PROGRAM POUNCPowerOn
VAR
	fbXAxisPowerOn : MC_Power;
	fbXAxisDrive : MC_MoveRelative;
	DegreesToRelativeMovment_0: DegreesToRelativeMovment;
	movementBuffer : MC_BufferMode; 
	SetMaxRelativePoint : LREAL;
	SetMaxSteeringAngle : INT;
	inputAngle : INT;
	ExecuteMovement : BOOL;
	ExecuteMovement1 : BOOL;
	MC_MoveAbsolute_0: MC_MoveAbsolute;
	MC_Home_0: MC_Home;
	StartHoming: BOOL;
	endSW AT %I*: BOOL;
	HomingActive: BOOL;
	MC_Reset_0: MC_Reset;
	reset: BOOL;
	PositionToDegree_0: PositionToDegree;
END_VAR

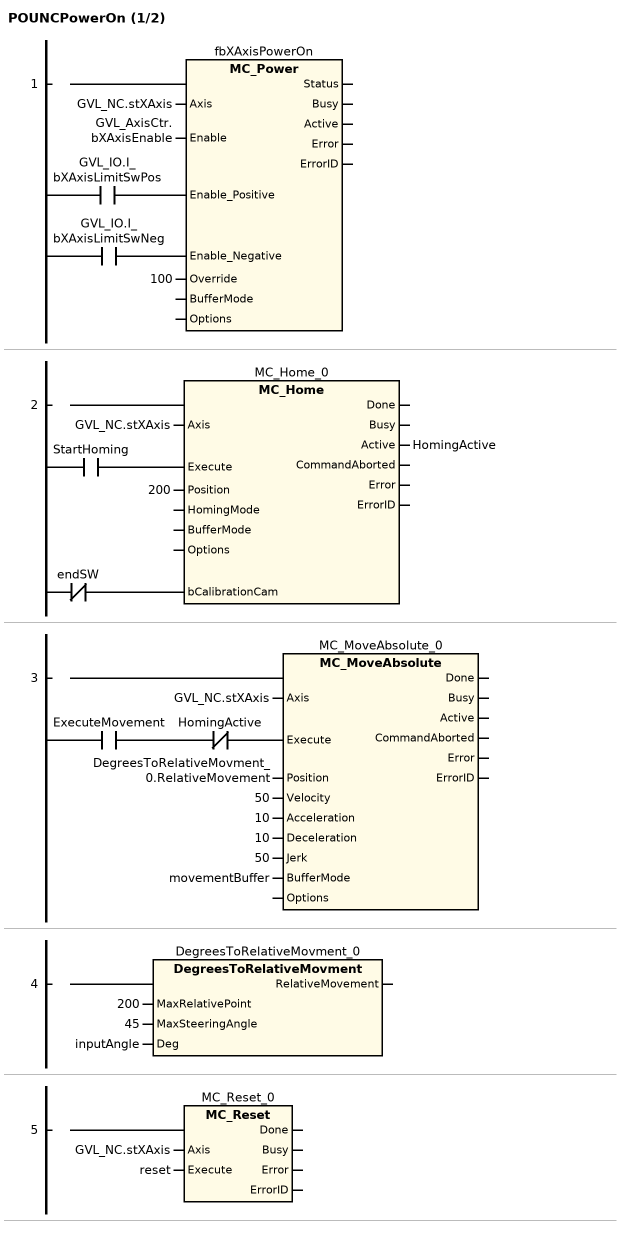
// NETWORK 1
fbXAxisPowerOn(
    Axis := GVL_NC.stXAxis,
    Enable := GVL_AxisCtr.bXAxisEnable,
    Enable_Positive := GVL_IO.I_bXAxisLimitSwPos,
    Enable_Negative := GVL_IO.I_bXAxisLimitSwNeg,
    Override := 100); // MC_Power

// NETWORK 2
MC_Home_0(
    Axis := GVL_NC.stXAxis,
    Execute := StartHoming,
    Position := 200,
    bCalibrationCam := NOT endSW,
    Active => HomingActive); // MC_Home

// NETWORK 3
MC_MoveAbsolute_0(
    Axis := GVL_NC.stXAxis,
    Execute := ExecuteMovement AND NOT HomingActive,
    Position := DegreesToRelativeMovment_0.RelativeMovement,
    Velocity := 50,
    Acceleration := 10,
    Deceleration := 10,
    Jerk := 50,
    BufferMode := movementBuffer); // MC_MoveAbsolute

// NETWORK 4
DegreesToRelativeMovment_0(MaxRelativePoint := 200, MaxSteeringAngle := 45, Deg := inputAngle); // DegreesToRelativeMovment

// NETWORK 5
MC_Reset_0(Axis := GVL_NC.stXAxis, Execute := reset); // MC_Reset

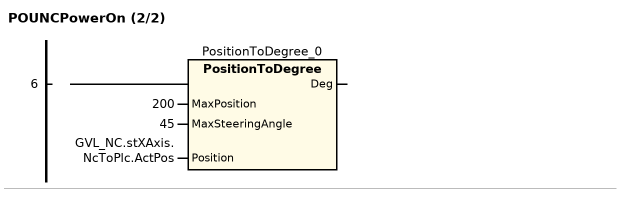
// NETWORK 6
PositionToDegree_0(MaxPosition := 200, MaxSteeringAngle := 45, Position := GVL_NC.stXAxis.NcToPlc.ActPos); // PositionToDegree

END_PROGRAM

(* stored: Version 1.1.0.1, ProductVersion 3.1.4024.3
   POU POUNCPowerOn: Id {518f66f2-a21f-4a9a-84b8-3594f5178ae2}, SpecialFunc None *)
